{attribute 'qualified_only'}
//{attribute 'strict'}
TYPE Drinks :
(
	Cola := 0,
	Fanta
);
END_TYPE

(* stored: Version 1.1.0.1, ProductVersion 3.1.4022.12
   DUT Drinks: Id {04b9c87a-fbd9-45c2-92b9-b51ca61fd7ab} *)
